FUNCTION_BLOCK PressureChamber_MNG
VAR_INPUT
	penningInt : INT;
	piraniInt : INT;
END_VAR
VAR_OUTPUT
	penningON : BOOL;
	pressureOut: REAL;
END_VAR
VAR
	voltage : REAL;
	penningPressure: REAL;
	piraniPressure: REAL;
	mix: REAL;
END_VAR

piraniPressure := ConvertPressure_Pirani(piraniInt);

IF piraniPressure > PARAM.PenningMix_Start THEN
	pressureOut := piraniPressure;
	penningON := FALSE;
ELSE
	penningON := TRUE;
	penningPressure := ConvertPressure_Penning(penningInt);
	mix := ( piraniPressure - PARAM.PenningMix_End ) / (PARAM.PenningMix_Start - PARAM.PenningMix_End);
	IF mix < 0 THEN
		mix := 0;
	END_IF
	pressureOut := mix * piraniPressure + ( 1 - mix) * penningPressure;
END_IF

END_FUNCTION_BLOCK

(* stored: Version 1.1.0.1, ProductVersion 3.1.4022.16
   POU PressureChamber_MNG: Id {689935d6-62b8-48d5-a1ed-4f695bb63735}, SpecialFunc None *)
